{attribute 'qualified_only'}
{attribute 'strict'}
TYPE eCapTestSTate :
(
	init 				:= 	0,
	WriteSerial			:=	1,
	WriteNameplateCap	:=	2,
	WriteDatetime		:=	3,
	StartSystem 		:= 	4,
	InitialCharge 		:= 	5,
	RestPeriod1			:= 	6,
	DischargeCycle 		:= 	7,
	RestPeriod2 		:= 	8,
	ChargeCycle 		:= 	9,
	RestPeriod3 		:= 	10,
	StopSystem  		:= 	11,
	done				:=	12
);
END_TYPE

(* stored: Version 1.1.0.1, ProductVersion 3.1.4026.18
   DUT eCapTestSTate: Id {949cd478-781c-4bcb-a384-ffef6bf0cd4e} *)
